// TwinCAT 3 PLC project PLC01
// ProgramVersion: 3.1.4023.0
// libraries:
//   Tc2_IoFunctions, * (Beckhoff Automation GmbH)
//   Tc2_Standard, * (Beckhoff Automation GmbH)
//   Tc2_System, * (Beckhoff Automation GmbH)
//   Tc2_Utilities, * (Beckhoff Automation GmbH)
//   Tc3_Module, * (Beckhoff Automation GmbH)
// project tree:
//   DUTs/Astrour/ FB_AstroUr.TcPOU
//   DUTs/Astrour/Functions/ fc_Day_Of_Year.TcPOU, fc_DEG.TcPOU, fc_DST.TcPOU, fc_Floor2.TcPOU, fc_Hour_To_Time.TcPOU, fc_Houre_To_TOD.TcPOU, fc_MODR.TcPOU, fc_RAD.TcPOU, fc_Set_Date.TcPOU, fc_Set_DT.TcPOU, fc_Sun_Midday.TcPOU, fc_Year_Of_Date.TcPOU
//   DUTs/Helgdag/ FB_SwedishHolidays.TcPOU
//   DUTs/Helgdag/Old/ FB_SwedishHolidaysOLD.TcPOU, POU_EasterDay.TcPOU
//   DUTs/KOH/ FB_KOH.TcPOU
//   DUTs/PID/ FB_PID.TcPOU
//   DUTs/Rampfunktion/ FB_Ramp.TcPOU
//   DUTs/Scale/ FB_Scale.TcPOU
//   DUTs/Select/ FB_Sel.TcPOU
//   DUTs/System/ FB_SystemTime.TcPOU, FB_TimerPulseSec.TcPOU, F_PLC_MS.TcPOU
//   DUTs/Tidkanal/ FB_TidKanalDrift.TcPOU
//   GVLs/ SYSTEM.TcGVL
//   / PlcTask.TcTTO
//   POUs/ MAIN.TcPOU
// real-time tasks:
//   TASK PlcTask: cycle T#10ms, priority 20, ADS port 350

CONFIGURATION PLC01
    RESOURCE PLC ON TwinCAT3
        TASK PlcTask(INTERVAL := T#10ms, PRIORITY := 20);
        PROGRAM MAIN WITH PlcTask : MAIN;
    END_RESOURCE
END_CONFIGURATION

// ---- GVLs/SYSTEM.TcGVL
{attribute 'qualified_only'}
VAR_GLOBAL
	nAliveCounter					: SINT; 			// PLC alive counter
    sDateAndTime					: STRING;			// Time and date
	dtSystemTime					: DATE_AND_TIME;	// Date and time
    uiYear							: UINT;				// Systemtime Year
    uiMonth							: UINT;				// Systemtime Month
    uiDayOfWeek 					: UINT;				// Systemtime Day of week
    uiDay							: UINT;				// Systemtime Day
    uiHour							: UINT;				// Systemtime Hour
    uiMinute						: UINT;				// Systemtime Minute
    uiSecond						: UINT;				// Systemtime Second
    uiMillisecond					: UINT;				// Systemtime Millisecond
    uiHourMinute					: UINT;				// Systemtime HourAndMinute
    dtDate							: DATE_AND_TIME;	// Variable for date and time
    uiTasktime						: UDINT;			// Tasktime
    uisystemtime 					: UDINT;			// System time	
    stTimeStruct					: TIMESTRUCT; 		// Timestruct
    sActTime						: STRING;			// Actual time
    uiSeconds						: UDINT;			// Variable for time in seconds
    bPowerFailDetect				: BOOL;				// Powerfail from UPS
    bIOError						: BOOL;				// IO-Error 
    bSavePersistentData				: BOOL;				// Saves persistent data manually              		
	tPlcUptime						: TIME;             // Last time PLC restart        		
	bWatchdogAlarm					: BOOL;				// Triggered watchdog alarm
	bWatchdogIsOK					: BOOL;				// Watchdog is ok  	
	bStartUp1s						: BOOL;				// Startup delay 1s after restart of TwinCAT
	bStartUp5s						: BOOL;				// Startup delay 5s after restart of TwinCAT
	bStartUp10s						: BOOL;				// Startup delay 10s after restart of TwinCAT
	bStartUp15s						: BOOL;				// Startup delay 15s after restart of TwinCAT
	bStartUp20s						: BOOL;				// Startup delay 20s after restart of TwinCAT
	bStartUp25s						: BOOL;				// Startup delay 25s after restart of TwinCAT
	bStartUp30s						: BOOL;				// Startup delay 30s after restart of TwinCAT
	bStartUp45s						: BOOL;				// Startup delay 45s after restart of TwinCAT
	bStartUp60s						: BOOL;				// Startup delay 60s after restart of TwinCAT
	bStartUp120s					: BOOL;				// Startup delay 120s after restart of TwinCAT
	bBurglarAlarmActive				: BOOL;				// Aktivt inbrottslarm 
	rOutdoorTemperature				: REAL;				// Outdoor temperature
	rAverageOutdoorTemperature		: REAL;				// Outdoor average temperature
	rAverageMinOutdoorTemperature	: REAL;				// Outdoor average min temperature	
	rAverageMaxOutdoorTemperature	: REAL;				// Outdoor average max temperature	
	rAverageIndoorTemperature		: REAL;				// Indoor average temperature
	bSummerCondition				: BOOL;        		// Summer condition active
	rCalculatedDewpoint				: REAL;				// Dewpoint   		          	

	sSystemID						: STRING;			// Current System ID
	sHostName						: STRING;			// Current hostname
	sAMSNetID						: STRING;			// Current AMS net ID
	sTargetType						: STRING;           
	sHardwareModel 					: STRING;
	sHardwareSerialNumber			: STRING;
	sHardwareVersion 				: STRING;
	sHardwareDate					: STRING;
	sHardwareCPU 					: STRING;
	sImageDevice					: STRING;
	sImageVersion 					: STRING;
	sImageLevel 					: STRING;
	sImageOsName 					: STRING;
	sImageOsVersion 				: STRING;
	sTwinCATVersion 				: STRING;
	sTwinCATRevision 				: STRING;
	sTwinCATBuild 					: STRING;
	sTwinCATLevel					: STRING;
	udiCpuUsage						: UDINT;	
	iArrWildCards					: ARRAY [0..100] OF INT;
	bArrWildCards					: ARRAY [0..100] OF BOOL;	
	
	
END_VAR

// ---- POUs/MAIN.TcPOU
PROGRAM MAIN
VAR
	fbTimeChannel 				: FB_TidkanalDrift;	
	fbAstroUr					: FB_AstroUr;
	fbSystemTime 				: FB_SystemTime;
	fbSwedishHolidays			: FB_SwedishHolidays;
	fbKOHFunction				: FB_KOH;
	
	bActivateTimeChannel		: BOOL; // Detta är en kommentar
	wMondayStartTime 			: WORD; // Detta är en kommentar
	wMondayStopTime 			: WORD; // Detta är en kommentar
	wTuesdayStartTime 			: WORD; // Detta är en kommentar
	wTuesdayStopTime 			: WORD; // Detta är en kommentar
	wWednesdayStartTime 		: WORD; // Detta är en kommentar
	wWednesdayStopTime 			: WORD; // Detta är en kommentar
	wThursdayStartTime 			: WORD; // Detta är en kommentar
	wThursdayStopTime 			: WORD; // Detta är en kommentar
	wFridayStartTime 			: WORD; // Detta är en kommentar
	wFridayStopTime 			: WORD; // Detta är en kommentar
	wSaturdayStartTime 			: WORD; // Detta är en kommentar
	wSaturdayStopTime 			: WORD; // Detta är en kommentar
	wSundayStartTime 			: WORD; // Detta är en kommentar
	wSundayStopTime 			: WORD; // Detta är en kommentar
	bTimeChannelActive			: BOOL; // Detta är en kommentar
	bSommarTidAktiv				: BOOL; // Detta är en kommentar
	bDetArMorktUteJustNu		: BOOL; // Detta är en kommentar
	strSoluppgang				: STRING; // Detta är en kommentar
	strSolnedgang				: STRING; // Detta är en kommentar
	//dActDate					: DATE:= D#2025-3-19; 
	dActDate					: DATE_AND_TIME; 
	dtTheDateAndTime			: DATE_AND_TIME;
	
	bLangfredagACT				: BOOL;
	bSkartorsdagACT				: BOOL;
	bPaskDagenACT				: BOOL;
	bPaskaftonACT				: BOOL;
	bAnnanDagPaskACT			: BOOL;
	bKristihimmelACT			: BOOL;
	bPingstAftonACT				: BOOL;
	bPingstDagenACT				: BOOL;
	bMidsommarDagenACT			: BOOL;
	bMidsommarAftonACT			: BOOL;
	bHalloweenACT				: BOOL;
	bJulaftonACT				: BOOL;
	bJuldagenACT				: BOOL;
	bAnnandagjulACT				: BOOL;
	bTrettondagACT				: BOOL;
	bNyarsaftonACT				: BOOL;
	bNyarsdagenACT				: BOOL;
	bForstamajACT				: BOOL;
	bNationaldagACT				: BOOL;
	bHelgDagAktivACT 			: BOOL;
	bAny						: BOOL; 
	iDay						: INT;
	
	// koh	
	bVarEnableKOHFunction		: BOOL;
	bVarBlockKOHFunction		: BOOL;
	bVarExceptionKOH			: BOOL;
	wVarMondayOn				: WORD;
	wVarMondayOff				: WORD;
	wVarTuesdayOn				: WORD;
	wVarTuesdayOff				: WORD;
	wVarWednesdayOn				: WORD;
	wVarWednesdayOff			: WORD;
	wVarThursdayOn				: WORD;
	wVarThursdayOff				: WORD;
	wVarFridayOn				: WORD;
	wVarFridayOff				: WORD;
	wVarSaturdayOn				: WORD;
	wVarSaturdayOff				: WORD;
	wVarSundayOn				: WORD;
	wVarSundayOff 				: WORD;
	diVarSystemCalcSetpoint 	: DINT;
	diVarDownRampTime  			: DINT;
	diVarSPEveningReduction 	: DINT;
	diVarSPWeekendReduction 	: DINT;
	diVarSPHolidayReduction 	: DINT;
	diVarSPExceptionReduction  	: DINT;
	diVarActualAverageRoomTemp 	: DINT;
	diVarAllowedMinRoomTemp  	: DINT;
	bVarKOHActive 				: BOOL;
	bVarKOHBlocked 				: BOOL;
	bVarAlarmBlocked			: BOOL;
	bVarAlarmMinTemp 			: BOOL;
	diVarKOHCalcOffset 			: DINT;
	bVarRampTimeActive			: BOOL;
	
END_VAR

VAR PERSISTENT	
	rLatitudeOrebro				: REAL; // Detta är en kommentar
	rLongitudeOrebro			: REAL; // Detta är en kommentar
	iOffsetSoluppgang			: INT; // Detta är en kommentar
	iOffsetSolnedgang			: INT; // Detta är en kommentar
END_VAR

fbSystemTime();
POU_EasterDay();

fbTimeChannel(
	bEn:= 					bActivateTimeChannel, 
	wMondayOn:= 			wMondayStartTime, 
	wMondayOff:= 			wMondayStopTime, 
	wTuesdayOn:= 			wTuesdayStartTime, 
	wTuesdayOff:= 			wTuesdayStopTime, 
	wWednesdayOn:= 			wWednesdayStartTime, 
	wWednesdayOff:= 		wWednesdayStopTime, 
	wThursdayOn:= 			wThursdayStartTime, 
	wThursdayOff:= 			wThursdayStopTime, 
	wFridayOn:= 			wFridayStartTime, 
	wFridayOff:= 			wFridayStopTime, 
	wSaturdayOn:= 			wSaturdayStartTime, 
	wSaturdayOff:= 			wSaturdayStopTime, 
	wSundayOn:= 			wSundayStartTime, 
	wSundayOff:= 			wSundayStopTime, 
	bOn=> 					bTimeChannelActive);

fbAstroUr(
	rLatitude:= 			rLatitudeOrebro, // Sätt latitud för platen du ska mäta på         
	rLongitude:= 			rLongitudeOrebro, // Sätt longitud för platsen du ska mäta på      
	iOffsetSunrise:= 		iOffsetSoluppgang, // Förskjut soluppgången här (teoretiskt)       
	iOffsetSunset:= 		iOffsetSolnedgang, // Förskjut solnedgången här (teoretiskt)       
	strSunrise=> 			strSoluppgang, // Detta är det förväntade klockslaget på soluppgång
	strSunset=> 			strSolnedgang, // Detta är det förväntade klockslaget på solnedgång
	bSummertime=> 			bSommarTidAktiv, // Det råder sommartid, åk till stranden          
	bDark=> 				bDetArMorktUteJustNu); // Är denna aktiv är det mörkt ute	         

fbSystemTime();
dActDate:=(fbSystemTime.dtSystemTime);

fbSwedishHolidays(
	dtActualDateAndTime=> 	dtTheDateAndTime, 
	bLangfredag=> 			bLangfredagACT, 
	bSkartorsdag=> 			bSkartorsdagACT, 
	bPaskDagen=> 			bPaskDagenACT, 
	bPaskafton=> 			bPaskaftonACT, 
	bAnnanDagPask=> 		bAnnanDagPaskACT, 
	bKristihimmel=> 		bKristihimmelACT, 
	bPingstAfton=> 			bPingstAftonACT, 
	bPingstDagen=> 			bPingstDagenACT, 
	bMidsommarDagen=> 		bMidsommarDagenACT, 
	bMidsommarAfton=> 		bMidsommarAftonACT, 
	bHalloween=> 			bHalloweenACT, 
	bJulafton=> 			bJulaftonACT, 
	bJuldagen=> 			bJuldagenACT, 
	bAnnandagjul=> 			bAnnandagjulACT, 
	bTrettondag=> 			bTrettondagACT, 
	bNyarsafton=> 			bNyarsaftonACT, 
	bNyarsdagen=> 			bNyarsdagenACT, 
	bForstamaj=> 			bForstamajACT, 
	bNationaldag=> 			bNationaldagACT, 
	bHelgDagAktiv=> 		bHelgDagAktivACT);


iDay:=fc_Day_Of_Year(IDATE:=TO_DATE (dActDate) );

	
	
fbKOHFunction(
	bEnableKOHFunction:= 			bVarEnableKOHFunction, 
	bBlockKOHFunction:= 			bVarBlockKOHFunction, 
	bExceptionKOH:= 				bVarExceptionKOH, 
	wMondayOn:= 					wVarMondayOn, 
	wMondayOff:= 					wVarMondayOff, 
	wTuesdayOn:= 					wVarTuesdayOn, 
	wTuesdayOff:= 					wVarTuesdayOff, 
	wWednesdayOn:= 					wVarWednesdayOn, 
	wWednesdayOff:= 				wVarWednesdayOff, 
	wThursdayOn:= 					wVarThursdayOn, 
	wThursdayOff:= 					wVarThursdayOff, 
	wFridayOn:= 					wVarFridayOn, 
	wFridayOff:= 					wVarFridayOff, 
	wSaturdayOn:= 					wVarSaturdayOn, 
	wSaturdayOff:= 					wVarSaturdayOff, 
	wSundayOn:= 					wVarSundayOn, 
	wSundayOff:= 					wVarSundayOff, 
	diSystemCalcSetpoint:= 			diVarSystemCalcSetpoint, 
	diDownRampTime:= 				diVarDownRampTime, 
	diSPEveningReduction:= 			diVarSPEveningReduction, 
	diSPWeekendReduction:= 			diVarSPWeekendReduction, 
	diSPHolidayReduction:= 			diVarSPHolidayReduction, 
	diSPExceptionReduction:= 		diVarSPExceptionReduction, 
	diActualAverageRoomTemp:= 		diVarActualAverageRoomTemp, 
	diAllowedMinRoomTemp:= 			diVarAllowedMinRoomTemp, 
	bKOHActive=> 					bVarKOHActive, 
	bKOHBlocked=> 					bVarKOHBlocked, 
	bAlarmBlocked=> 				bVarAlarmBlocked, 
	bAlarmMinTemp=> 				bVarAlarmMinTemp, 
	diKOHCalcOffset=> 				diVarKOHCalcOffset, 
	bRampTimeActive=> 				bVarRampTimeActive);

END_PROGRAM

// ---- DUTs/Tidkanal/FB_TidKanalDrift.TcPOU
FUNCTION_BLOCK FB_TidKanalDrift
VAR_INPUT
	bEn				: BOOL;		// Aktivera block
	wMondayOn		: WORD;		// Starttid Måndag
	wMondayOff		: WORD;		// Stopptid Måndag
	wTuesdayOn		: WORD;		// Starttid Tisdag
	wTuesdayOff		: WORD;		// Stopptid Tisdag
	wWednesdayOn	: WORD;		// Starttid Onsdag
	wWednesdayOff	: WORD;		// Stopptid Onsdag
	wThursdayOn		: WORD;		// Starttid Torsdag
	wThursdayOff	: WORD;		// Stopptid Torsdag
	wFridayOn		: WORD;		// Starttid Fredag
	wFridayOff		: WORD;		// Stopptid Fredag
	wSaturdayOn		: WORD;		// Starttid Lördag
	wSaturdayOff	: WORD;		// Stopptid Lördag
	wSundayOn		: WORD;		// Starttid Söndag
	wSundayOff		: WORD;		// Stopptid Söndag
END_VAR
	
VAR_OUTPUT
	bOn				: BOOL;		// Tidkanal aktiv
END_VAR


VAR
	fbSystemTime 	: FB_SystemTime;
END_VAR

// Tidkanal
fbSystemTime();
IF bEN THEN

CASE fbSystemTime.nWeekDay OF
	
		1: // Måndag 
		IF wMondayOff < wMondayOn THEN
			// 22:00-03:00
			IF fbSystemTime.nHourMinute >= wMondayOn OR fbSystemTime.nHourMinute < wMondayOff THEN
				bOn := TRUE;
			ELSE
				bOn := FALSE;
			END_IF
		ELSE
			// 06:00-22:00	
			IF fbSystemTime.nHourMinute >= wMondayOn AND fbSystemTime.nHourMinute < wMondayOff THEN
				bOn := TRUE;
			ELSE
				bOn := FALSE;
			END_IF
		END_IF	
		
		2: // Tisdag
		IF wTuesdayOff < wTuesdayOn THEN
			// 22:00-03:00
			IF fbSystemTime.nHourMinute >= wTuesdayOn OR fbSystemTime.nHourMinute < wTuesdayOff THEN
				bOn := TRUE;
			ELSE
				bOn := FALSE;
			END_IF
		ELSE
			// 06:00-22:00	
			IF fbSystemTime.nHourMinute >= wTuesdayOn AND fbSystemTime.nHourMinute < wTuesdayOff THEN
				bOn := TRUE;
			ELSE
				bOn := FALSE;
			END_IF
		END_IF		
		
		3: // Onsdag
		IF wWednesdayOff < wWednesdayOn THEN
			// 22:00-03:00
			IF fbSystemTime.nHourMinute >= wWednesdayOn OR fbSystemTime.nHourMinute < wWednesdayOff THEN
				bOn := TRUE;
			ELSE
				bOn := FALSE;
			END_IF
		ELSE
			// 06:00-22:00	
			IF fbSystemTime.nHourMinute >= wWednesdayOn AND fbSystemTime.nHourMinute < wWednesdayOff THEN
				bOn := TRUE;
			ELSE
				bOn := FALSE;
			END_IF
		END_IF	
		
		4: // Torsdag
		IF wThursdayOff < wThursdayOn THEN
			// 22:00-03:00
			IF fbSystemTime.nHourMinute >= wThursdayOn OR fbSystemTime.nHourMinute < wThursdayOff THEN
				bOn := TRUE;
			ELSE
				bOn := FALSE;
			END_IF
		ELSE
			// 06:00-22:00	
			IF fbSystemTime.nHourMinute >= wThursdayOn AND fbSystemTime.nHourMinute < wThursdayOff THEN
				bOn := TRUE;
			ELSE
				bOn := FALSE;
			END_IF
		END_IF	

		5: // Fredag 
		IF wFridayOff < wFridayOn THEN
			// 22:00-03:00
			IF fbSystemTime.nHourMinute >= wFridayOn OR fbSystemTime.nHourMinute < wFridayOff THEN
				bOn := TRUE;
			ELSE
				bOn := FALSE;
			END_IF
		ELSE
			// 06:00-22:00	
			IF fbSystemTime.nHourMinute >= wFridayOn AND fbSystemTime.nHourMinute < wFridayOff THEN
				bOn := TRUE;
			ELSE
				bOn := FALSE;
			END_IF
		END_IF	
		
		6: // Lördag
		IF wSaturdayOff < wSaturdayOn THEN
			// 22:00-03:00
			IF fbSystemTime.nHourMinute >= wSaturdayOn OR fbSystemTime.nHourMinute < wSaturdayOff THEN
				bOn := TRUE;
			ELSE
				bOn := FALSE;
			END_IF
		ELSE
			// 06:00-22:00	
			IF fbSystemTime.nHourMinute >= wSaturdayOn AND fbSystemTime.nHourMinute < wSaturdayOff THEN
				bOn := TRUE;
			ELSE
				bOn := FALSE;
			END_IF
		END_IF	
		
		0: // Söndag
		IF wSundayOff < wSundayOn THEN
			// 22:00-03:00
			IF fbSystemTime.nHourMinute >= wSundayOn OR fbSystemTime.nHourMinute < wSundayOff THEN
				bOn := TRUE;
			ELSE
				bOn := FALSE;
			END_IF
		ELSE
			// 06:00-22:00	
			IF fbSystemTime.nHourMinute >= wSundayOn AND fbSystemTime.nHourMinute < wSundayOff THEN
				bOn := TRUE;
			ELSE
				bOn := FALSE;
			END_IF
		END_IF
END_CASE


ELSE bOn := FALSE;
	
END_IF

END_FUNCTION_BLOCK

// ---- DUTs/System/FB_SystemTime.TcPOU
(*
:Beskrivning:	| Läser systemtiden.
:Instruktioner:	| Ändra sAMSNetID för annan tidsserver. Lämna tom för lokal tid i PLC.

:Versionshistorik:
+-------------+------------+----------------+------------+------------------------------------------+
|Datum        | Version    | Skapad under   | Författare | Kommentar                                |
+=============+============+================+============+==========================================+
|2020-02-20   | 1.0.0.1    | V3.1.4022.30   | CMC dev.   | Funktionsblock skapat                    |
+-------------+------------+----------------+------------+------------------------------------------+
	
*)
FUNCTION_BLOCK FB_SystemTime
VAR_INPUT
	sAMSNetID			: STRING:='';	// AMSNet-ID
END_VAR

VAR_OUTPUT
	dtSystemTime		: DT;			// Systemtid
	bGetTimeBusy		: BOOL;			// Busy  		
	bGetTimeError		: BOOL;			// Error
	nGetTimeErrorCode	: UDINT;		// ErrorID
	nYear				: DWORD;		// År
	nMonth				: DWORD;		// Månad
	nDay				: DWORD;		// Dag
	nWeekDay 			: DWORD;		// Veckodag
	nHour				: DWORD;		// Timme
	nMinute 			: DWORD;		// Minut
	nSecond				: DWORD;		// Sekund
	nMilliSecond		: DWORD;		// Millisekund
	nHourMinute			: DWORD;		// Timme och minut (HHMM)
END_VAR

VAR
	fbGetTime			: NT_GetTime;
	fbTimerPulseSec		: FB_TimerPulseSec;
END_VAR

fbTimerPulseSec(bStart := TRUE, nTime := 5); // FB_TimerPulseSec
fbGetTime(NETID := sAMSNetID, START := fbTimerPulseSec.bPulse, TMOUT := T#5s); // NT_GetTime
bGetTimeBusy := fbGetTime.BUSY;
bGetTimeError := fbGetTime.ERR;
nGetTimeErrorCode := fbGetTime.ERRID;
dtSystemTime := SYSTEMTIME_TO_DT(TIMESTR := fbGetTime.TIMESTR);
nYear := TO_DWORD(fbGetTime.TIMESTR.wYear);
nMonth := TO_DWORD(fbGetTime.TIMESTR.wMonth);
nDay := TO_DWORD(fbGetTime.TIMESTR.wDay);
nWeekDay := TO_DWORD(fbGetTime.TIMESTR.wDayOfWeek);
nHour := TO_DWORD(fbGetTime.TIMESTR.wHour);
nMinute := TO_DWORD(fbGetTime.TIMESTR.wMinute);
nSecond := TO_DWORD(fbGetTime.TIMESTR.wSecond);
nMilliSecond := TO_DWORD(fbGetTime.TIMESTR.wMilliseconds);
nHourMinute := nHour * 100 + nMinute;

END_FUNCTION_BLOCK

// ---- DUTs/System/FB_TimerPulseSec.TcPOU
(*
:Beskrivning:	| Timern är igång så länge bStart är hög. bPulse pulsar när bStart går från FALSE till TRUE och när nTIME är uppnådd. När nTIME är uppnådd börjar timern räkna om.
:Instruktioner:	|  

:Versionshistorik:
+-------------+------------+----------------+------------+------------------------------------------+
|Datum        | Version    | Skapad under   | Författare | Kommentar                                |
+=============+============+================+============+==========================================+
|2020-02-21   | 1.0.0.1    | V3.1.4022.30   | CMC dev.   | Funktionsblock skapat					|
+-------------+------------+----------------+------------+------------------------------------------+
	
*)
FUNCTION_BLOCK FB_TimerPulseSec
VAR_INPUT
	bStart 		: BOOL;  	// Aktivera timer
	nTIME		: DWORD; 	// Tid mellan pulserna (s)
END_VAR

VAR_OUTPUT
	bPulse		: BOOL; 	// Pulsutgång
END_VAR

VAR
	Start		: BOOL;
	init		: BOOL;
	tx			: DWORD;
	last		: DWORD;
	ms			: DWORD;
	Sec			: UDINT;
	
	R_TRIG		: R_TRIG;
END_VAR

(*

Information om block:

Källa: Oscat OnTime

*)

// Read system time
tx := F_PLC_MS();

// Make sure the first cycle works correctly
IF NOT init OR NOT bStart THEN
	init := TRUE;
	ms := 0;
ELSIF bStart THEN
	// Add the current milliseconds
	ms := (tx - last) + ms;
	IF ms >= 100 THEN
		Sec := Sec + 1;
		ms := ms - 100;
	END_IF
END_IF

IF NOT bStart THEN
	Sec := 0;
END_IF
last := tx;

IF bStart AND NOT Start THEN
	R_TRIG(CLK := bStart, Q => bPulse);
	Start := TRUE;
ELSIF bStart AND Sec >= TO_UDINT(nTIME) THEN
	bPulse := TRUE;
	Sec := 0;
ELSIF bStart THEN	
	bPulse := FALSE;
	Sec := Sec;
ELSE
	bPulse := FALSE;
	Start := FALSE;
	R_TRIG(CLK := FALSE);
END_IF

END_FUNCTION_BLOCK

// ---- DUTs/System/F_PLC_MS.TcPOU
(*
:Beskrivning:	| Hämtar PLCns interna timer i Millisekunder.
:Instruktioner:	|  

:Versionshistorik:
+-------------+------------+----------------+------------+-------------------------------------------+
|Datum        | Version    | Skapad under   | Författare | Kommentar                                 |
+=============+============+================+============+===========================================+
|2020-02-21   | 1.0.0.1    | V3.1.4022.30   | CMC dev.   | Funktion skapad							 |
+-------------+------------+----------------+------------+-------------------------------------------+
	
*)
FUNCTION F_PLC_MS : DWORD;	// Millisekunder
VAR CONSTANT
	N 			: INT := 0;
	debug		: BOOL := 0;
	offset		: DWORD := 0;
END_VAR
VAR
	tx		 	: TIME;		// Timer i Millisekunder
END_VAR

(*

Information om block:

Källa: Oscat T_PLC_MS

*)

tx := TIME();
F_PLC_MS := TIME_TO_DWORD(Tx);

IF debug THEN
	F_PLC_MS := (SHL(F_PLC_MS,N) OR SHL(DWORD#1,N)-1) + OFFSET;
END_IF;

END_FUNCTION

// ---- DUTs/Astrour/FB_AstroUr.TcPOU
FUNCTION_BLOCK FB_AstroUr

VAR_INPUT
	rLatitude 				: REAL; // Latitud där anläggningen befinner sig
	rLongitude 				: REAL; // Longitud där anläggningen befinner sig
	iOffsetSunrise			: DINT;	// Offset för soluppgång i minuter
	iOffsetSunset			: DINT;	// Offset för solnedgång i minuter
END_VAR         			
                			
VAR_OUTPUT      			
	strSunrise				: STRING(5); // SunRise som string
	strSunset				: STRING(5); // Sunset som string
	bSummertime				: BOOL; // Indikering sommartid
	bDark					: BOOL; // Indikering solen har gått ner
END_VAR

VAR
	fbSystemTime 			: FB_SystemTime;
	                		
	dDate 					: DATE; // Aktuellt datum
	rSunPosMidday			: REAL; // Solens position mitt på dagen
	tDelta					: TIME; // Dela, tiden från mitt på dagen till soluppgång/nedgång
	rLatRad					: REAL; // Latitud omberäknad till radianer
	todActSunRise 			: TOD; // Soluppgång aktuell dag
	todActSunSet 			: TOD; // Solnedgång aktuell dag
	todActTime				: TIME_OF_DAY; // Aktuellt klockslag	
	todMidDay				: TOD; // Aktuell middagstid (när solen står i Zenit)
	rSunAngleMidday 		: REAL; // Solens vinkel mitt på dagen	
	dwSunSet				: DWORD; // Mellanvariabel för konvertering
	dwSunRise				: DWORD; // Mellanvariabel för konvertering            	
	rHeightAngle			: REAL := -0.83333333333; // Solens tim-vinkel
	todSunRise				: TOD;
	todSunSet				: TOD;
	dtVarSystemTime 		: DATE_AND_TIME;
	todVarTimeOfDay			: TIME_OF_DAY;
	
	dwSunRiseMinute			: DWORD;
	dwSunRiseHour			: DWORD;
	dwSunRiseTime			: DWORD;
	
	dwSunSetMinute			: DWORD;
	dwSunSetHour			: DWORD;
	dwSunSetTime			: DWORD;
	
	strHourSunRise			: STRING(2);
	strMinuteSunRise		: STRING(2);  
	strHourSunSet			: STRING(2);
	strMinuteSunSet			: STRING(2);   
END_VAR

// Anrop och variabelhanteringar
fbSystemTime();

dtVarSystemTime:= 	fbSystemTime.dtSystemTime;
todActTime:= 		todVarTimeOfDay;
dDate:= 			TO_DATE(dtVarSystemTime);
todVarTimeOfDay:= 	TO_TOD (fbSystemTime.dtSystemTime); 
rLatRad:=			rLatitude * 0.0174532925199433;
todMidDay:=			fc_Sun_Midday(rLongitude, dDate);

// Beräknar solposition
rSunPosMidday := 0.40954 * SIN(0.0172 * (INT_TO_REAL(fc_Day_Of_Year(dDate)) - 79.35));
rSunAngleMidday := fc_DEG(rSunPosMidday);

// Sätter solvinkel
IF rSunAngleMidday > 180.0 THEN
	rSunAngleMidday := rSunAngleMidday - 360.0;
END_IF;

rSunAngleMidday := 90.0 - rLatitude + rSunAngleMidday;

// Beräknar tid mellan solens högsta punkt och solnedgång resp. soluppgång
tDelta := fc_Hour_To_Time(ACOS((SIN(fc_RAD(rHeightAngle)) - SIN(rLatRad) * SIN(rSunPosMidday)) / (COS(rLatRad) * COS(rSunPosMidday))) * 3.819718632);

todActSunRise := todMidDay - tDelta;
todActSunSet := todMidDay + tDelta;

// Sommartid eller ej 
bSummertime := fc_DST(UTC:= dtVarSystemTime);

// Förskjutning om sommartid råder
IF bSummertime THEN
	todSunRise 	:= todActSunRise + T#2H + DINT_TO_TIME(iOffsetSunrise * 60000);
	todSunSet	:= todActSunSet  + T#2H + DINT_TO_TIME(iOffsetSunset  * 60000); ELSE
	todSunRise 	:= todActSunRise + T#1H + DINT_TO_TIME(iOffsetSunrise * 60000);
	todSunSet	:= todActSunSet  + T#1H + DINT_TO_TIME(iOffsetSunset  * 60000);
END_IF

// Sätter bool om det är mörkt ute
IF (todSunRise > todActTime) OR (todSunSet < todActTime) THEN
	bDark := TRUE; ELSE
	bDark := FALSE;	
END_IF

// Skapar STRING för att presentera soluppgång / solnedgång i SCADA/KOD

// Soluppgång
dwSunRiseHour:= TOD_TO_DWORD(todSunRise)/3600000;
dwSunRiseMinute:= TOD_TO_DWORD(todSunRise)/60000;
dwSunRiseTime:= dwSunRiseMinute -(60 * dwSunRiseHour);

IF dwSunRiseHour < 10 THEN
	strHourSunRise := concat ('0',DWORD_TO_STRING(dwSunRiseHour)); ELSE
	strHourSunRise := DWORD_TO_STRING(dwSunRiseHour);	
END_IF

IF dwSunRiseTime < 10 THEN 
	strMinuteSunRise := concat('0',DWORD_TO_STRING(dwSunRiseTime)); ELSE
	strMinuteSunRise := DWORD_TO_STRING(dwSunRiseTime);
END_IF

// Solnedgång
dwSunSetHour:= TOD_TO_DWORD(todSunSet)/3600000;
dwSunSetMinute:= TOD_TO_DWORD(todSunSet)/60000;
dwSunSetTime:= dwSunSetMinute -(60 * dwSunSetHour);

IF dwSunSetHour < 10 THEN
	strHourSunSet := concat ('0',DWORD_TO_STRING(dwSunSetHour)); ELSE
	strHourSunSet := DWORD_TO_STRING(dwSunSetHour);	
END_IF

IF dwSunSetMinute < 10 THEN 
	strMinuteSunSet := concat('0',DWORD_TO_STRING(dwSunSetTime)); ELSE
	strMinuteSunSet := DWORD_TO_STRING(dwSunSetTime);
END_IF

// Klara strängar
strSunRise:= concat(strHourSunRise,':');
strSunRise:= concat(strSunRise, strMinuteSunRise);
strSunSet:= concat(strHourSunSet,':');
strSunSet:= concat(strSunSet, strMinuteSunSet);

END_FUNCTION_BLOCK

// ---- DUTs/Astrour/Functions/fc_Sun_Midday.TcPOU
FUNCTION fc_Sun_Midday : TOD
VAR_INPUT
	LON : REAL;
	UTC : DATE;
END_VAR
VAR
	T 		: REAL;
	OFFSET 	: REAL;
END_VAR

T := INT_TO_REAL(fc_Day_Of_Year(utc));


OFFSET := -0.1752 * SIN(0.033430 * T + 0.5474) - 0.1340 * SIN(0.018234 * T - 0.1939);
fc_Sun_Midday := fc_Houre_To_TOD(12.0 - OFFSET - lon * 0.0666666666666);

END_FUNCTION

// ---- DUTs/Astrour/Functions/fc_Day_Of_Year.TcPOU
FUNCTION fc_Day_Of_Year : int
VAR_INPUT
		IDATE : DATE;
END_VAR
VAR
END_VAR


fc_Day_Of_Year := UDINT_TO_INT((DATE_TO_UDINT(idate) / UDINT#86400) MOD UDINT#1461);

IF fc_Day_Of_Year > 729 THEN
	IF fc_Day_Of_Year > 1095 THEN fc_Day_Of_Year := fc_Day_Of_Year - 1095; ELSE fc_Day_Of_Year := fc_Day_Of_Year - 729; END_IF;
ELSIF fc_Day_Of_Year > 364 THEN
	fc_Day_Of_Year := fc_Day_Of_Year - 364;
ELSE
	fc_Day_Of_Year := fc_Day_Of_Year + 1;
END_IF;

END_FUNCTION

// ---- DUTs/Astrour/Functions/fc_Houre_To_TOD.TcPOU
FUNCTION fc_Houre_To_TOD : TOD
VAR_INPUT
		IN : REAL;
END_VAR
VAR
END_VAR

fc_Houre_To_TOD := DWORD_TO_TOD(REAL_TO_DWORD(IN * 3600000));

END_FUNCTION

// ---- DUTs/Astrour/Functions/fc_DEG.TcPOU
FUNCTION fc_DEG : real
VAR_INPUT
		rad : REAL;
END_VAR
VAR
END_VAR

fc_DEG := fc_MODR(57.29577951308232 * RAD, 360.0);

END_FUNCTION

// ---- DUTs/Astrour/Functions/fc_MODR.TcPOU
FUNCTION fc_MODR : real
VAR_INPUT
	IN : REAL;
	DIVI : REAL;
END_VAR
VAR
END_VAR

IF divi = 0.0 THEN
	fc_MODR := 0.0;
ELSE
	fc_MODR := in - DINT_TO_REAL(fc_Floor2(in / divi)) * divi;
END_IF;

END_FUNCTION

// ---- DUTs/Astrour/Functions/fc_Floor2.TcPOU
FUNCTION fc_Floor2 : DINT
VAR_INPUT
	X : REAL;
END_VAR
VAR
END_VAR

fc_Floor2 := REAL_TO_DINT(X);
IF DINT_TO_REAL(fc_Floor2) > X THEN
	fc_Floor2 := fc_Floor2 - 1;
END_IF;

END_FUNCTION

// ---- DUTs/Astrour/Functions/fc_Hour_To_Time.TcPOU
FUNCTION fc_Hour_To_Time : Time
VAR_INPUT
		IN : REAL;
END_VAR
VAR
END_VAR

fc_Hour_To_Time := DWORD_TO_TIME(REAL_TO_DWORD(IN * 3600000));

END_FUNCTION

// ---- DUTs/Astrour/Functions/fc_RAD.TcPOU
FUNCTION fc_RAD : real
VAR_INPUT
	DEG : REAL;
END_VAR
VAR
END_VAR

fc_RAD := fc_MODR(0.0174532925199433 * DEG, 6.28318530717958647692528676655900576);

END_FUNCTION

// ---- DUTs/Astrour/Functions/fc_DST.TcPOU
FUNCTION fc_DST : bool
VAR_INPUT
	UTC 	: DT;
END_VAR
VAR
	yr 		: INT;
	yr4 	: DWORD;
	ltc		: DWORD;
	idate 	: DWORD;
END_VAR

yr := fc_Year_Of_Date(DT_TO_DATE(UTC));
ltc := DT_TO_DWORD(UTC);
idate := DT_TO_DWORD(fc_Set_DT(yr, 3, 31, 1, 0, 0));
yr4 := SHR(5 * INT_TO_DWORD(yr), 2) + 1;
fc_DST := (idate - ((yr4 + 3) MOD 7) * 86400 <= ltc) AND (idate + (214 - (yr4) MOD 7) * 86400 > ltc);

END_FUNCTION

// ---- DUTs/Astrour/Functions/fc_Year_Of_Date.TcPOU
FUNCTION fc_Year_Of_Date : INT
VAR_INPUT
		IDATE : DATE;
END_VAR
VAR
END_VAR

fc_Year_Of_Date := DWORD_TO_INT((DATE_TO_DWORD(idate) + 43200) / 31557600 + 1970);

END_FUNCTION

// ---- DUTs/Astrour/Functions/fc_Set_DT.TcPOU
FUNCTION fc_Set_DT : DT
VAR_INPUT
	year 	: INT;
	month 	: INT;
	day 	: INT;
	hour 	: INT;
	minute 	: INT;
	second 	: INT;
END_VAR
VAR
END_VAR

fc_Set_DT := DWORD_TO_DT(DATE_TO_DWORD(fc_Set_Date(YEAR, MONTH, day)) + INT_TO_DWORD(SECOND) + INT_TO_DWORD(MINUTE) * 60 + INT_TO_DWORD(HOUR) * 3600);

END_FUNCTION

// ---- DUTs/Astrour/Functions/fc_Set_Date.TcPOU
FUNCTION fc_Set_Date : date
VAR_INPUT
	YEAR 	: INT;
	MONTH 	: INT;
	DAY 	: INT;
END_VAR
VAR
	count 	: INT;
END_VAR

IF month > 2 THEN
	count := (month - 1) * 30;
	IF month > 7 THEN count := count + SHR(month - 3,1); ELSE count := count + SHR(month - 4,1); END_IF;
	(* chech for leap year and add one day if true *)
	IF SHL(year,14) = 0 THEN count := count + 1; END_IF;
ELSE
	count := (month - 1) * 31;
END_IF;

fc_Set_Date := DWORD_TO_DATE((INT_TO_DWORD(count + day - 1) + SHR(INT_TO_DWORD(year) * 1461 - 2878169, 2)) * 86400);

END_FUNCTION

// ---- DUTs/Helgdag/FB_SwedishHolidays.TcPOU
FUNCTION_BLOCK FB_SwedishHolidays
VAR_INPUT
END_VAR

VAR_OUTPUT
	dtActualDateAndTime			: DATE_AND_TIME;
	bLangfredag					: BOOL;
	bSkartorsdag				: BOOL;
	bPaskDagen					: BOOL;
    bPaskafton					: BOOL;
    bAnnanDagPask				: BOOL;
    bKristihimmel				: BOOL;
    bPingstAfton				: BOOL;
    bPingstDagen				: BOOL;
    bMidsommarDagen				: BOOL;
    bMidsommarAfton				: BOOL;
    bHalloween					: BOOL;
    bJulafton					: BOOL;
    bJuldagen					: BOOL;
    bAnnandagjul				: BOOL;
    bTrettondag					: BOOL;
    bNyarsafton					: BOOL;
    bNyarsdagen					: BOOL;
    bForstamaj					: BOOL;
    bNationaldag				: BOOL;
	bHelgDagAktiv				: BOOL;
END_VAR

VAR
	fbSystemTime 				: FB_SystemTime;
    iYear 						: INT; // Aktuellt år	
    iMonth						: INT;
	iDay						: INT;
    iEastermDayOfYear			: INT; // Påskdagens dagnummer i året
    isLeapYear 					: BOOL; // Flagga för skottår	
	stSystemTime				: TIMESTRUCT;
    arrMonthDays 				: ARRAY[1..12] OF INT := [31,28,31,30,31,30,31,31,30,31,30,31]; // Dagar per månad
    iDayOfYear					: INT;
    a, b, c, d, e, f, g, h, i, k, L, m, n : INT; // Variabler för Gauss algoritm
	iDayOfWeek					: INT;
	iActMonth					: INT;
	
	iVarHalloweenDay			: INT;
	iVarMidsommardagen 			: INT;
	iMidsommardagenDayOfYear	: INT;
	iVarMidsommardagenDayOfWeek	: INT;
	iVarMidsommardagen1			: INT;
	iSumDays					: INT;
	iVarDayOfYearCristmas		: INT;
	iVarDayForstamaj			: INT;
	iVarNationaldag				: INT;
	iVarJuldagen				: INT;
	
	iLangfredag					: INT;
 	iSkartorsdag				: INT;
	iPaskDagen					: INT;
 	iPaskafton					: INT;
 	iAnnanDagPask				: INT;
	iKristihimmel				: INT;
	iPingstAfton				: INT;
	iPingstDagen				: INT;
	iMidsommarDagen				: INT;
	iMidsommarAfton				: INT;
	iHalloween					: INT;
	iJulafton					: INT;
	iJuldagen					: INT;
	iAnnandagjul				: INT;
	iTrettondag					: INT;
    iNyarsafton					: INT;	
    iNyarsdagen					: INT;	
    iForstamaj					: INT;		
    iNationaldag				: INT;
END_VAR

VAR PERSISTENT
	iYear2000		: INT:=2000;
END_VAR

fbSystemTime();
iDayOfYear:= fc_Day_Of_Year(IDATE:=TO_DATE (fbSystemTime.dtSystemTime)) + 1;
iYear:= DWORD_TO_INT(fbSystemTime.nYear);
iDayOfWeek:= DWORD_TO_INT(fbSystemTime.nDay);
iActMonth:= TO_INT (fbSystemTime.nMonth);
dtActualDateAndTime:= (fbSystemTime.dtSystemTime);

// Gauss algoritm för att räkna ut påskdagen
a := iYear MOD 19;
b := iYear / 100;
c := iYear MOD 100;
d := b / 4;
e := b MOD 4;
f := (b + 8) / 25;
g := (b - f + 1) / 3;
h := (19 * a + b - d - g + 15) MOD 30;
i := c / 4;
k := c MOD 4;
L := (32 + 2 * e + 2 * i - h - k) MOD 7;
m := (a + 11 * h + 22 * L) / 451;
n := (h + L - 7 * m + 114);
iMonth := n / 31;
iDay := (n MOD 31) + 1;

// Kontrollera om året är skottår
IF (iYear MOD 4 = 0 AND iYear MOD 100 <> 0) OR (iYear MOD 400 = 0) THEN
    isLeapYear := TRUE;
    arrMonthDays[2] := 29; // Februari har 29 dagar i skottår
ELSE
    isLeapYear := FALSE;
END_IF

// Beräkna årets dag för påskdagen
iEastermDayOfYear := iDay; // Startvärde
FOR i := 1 TO iMonth - 1 DO
    iEastermDayOfYear := iEastermDayOfYear + arrMonthDays[i]; // Addera dagar i tidigare månader
END_FOR

// Beräkna årets dag för 31 oktober, Halloween
iVarHalloweenDay := 31; // Startvärde för Halloweens dag i oktober
FOR i := 1 TO 9 DO // Loopar igenom månaderna januari-september
    iVarHalloweenDay := iVarHalloweenDay + arrMonthDays[i]; // Addera dagar i tidigare månader
END_FOR


// 1. Beräkna veckodag för 20 juni enligt Zeller's Congruence
iVarMidsommardagenDayOfWeek := (20 + ((13 * 7) / 5) + (iYear MOD 100) + ((iYear MOD 100) / 4) + ((iYear / 100) / 4) - (2 * (iYear / 100))) MOD 7;

// 2. Konvertera från Zeller-format till Beckhoff-format (Söndag = 0, Måndag = 1, ..., Lördag = 6)
iVarMidsommardagenDayOfWeek := (iVarMidsommardagenDayOfWeek + 6) MOD 7;

// 3. Hitta första lördagen från och med 20 juni
IF iVarMidsommardagenDayOfWeek = 6 THEN
    iVarMidsommardagen := 20; // 20 juni är lördag
ELSE
    iVarMidsommardagen := 20 + ((6 - iVarMidsommardagenDayOfWeek) MOD 7);
END_IF

// 4. Beräkna årets dag (julianska kalenderdagar) inklusive skottår
iVarMidsommardagen1 := iVarMidsommardagen;

// Lägg till dagarna från januari till maj
iSumDays := 0;
FOR i := 1 TO 5 DO
    iSumDays := iSumDays + arrMonthDays[i];
END_FOR

// Om det är skottår, lägg till 1 dag efter februari
IF ((iYear MOD 4 = 0 AND iYear MOD 100 <> 0) OR (iYear MOD 400 = 0)) THEN
    iSumDays := iSumDays + 1;  // Flytta till här!
END_IF

iVarMidsommardagen1 := iVarMidsommardagen1 + iSumDays;


// Beräknar årets dag för 25 december
iVarDayOfYearCristmas := 24; // Startvärde för juldagen
FOR i := 1 TO 11 DO // Loopar igenom månaderna januari-november
    iVarDayOfYearCristmas := iVarDayOfYearCristmas + arrMonthDays[i]; // Addera dagar i tidigare månader
END_FOR

IF isLeapYear THEN
    iVarDayOfYearCristmas := iVarDayOfYearCristmas + 1;
END_IF

// Beräknar årets dag för 1 maj
iVarDayForstamaj := 0; // Startvärde för 1 maj
FOR i := 1 TO 4 DO // Loopar igenom månaderna januari-april *)
    iVarDayForstamaj := iVarDayForstamaj + arrMonthDays[i]; //Addera dagar i tidigare månader
END_FOR

IF isLeapYear THEN
    iVarDayForstamaj := iVarDayForstamaj + 1;
END_IF

// Beräkna sveriges nationaldag
iVarNationaldag := 5; // Startvärde för 6 juni
FOR i := 1 TO 5 DO // Loopar igenom månaderna januari-maj
    iVarNationaldag := iVarNationaldag + arrMonthDays[i]; // Addera dagar i tidigare månader
END_FOR
IF isLeapYear THEN
    iVarNationaldag := iVarNationaldag + 1;
END_IF


// Ger var värde för resp. dag
iLangfredag 		:= iEastermDayOfYear - 2;
iSkartorsdag	 	:= iEastermDayOfYear - 3;
iPaskDagen			:= iEastermDayOfYear;
iPaskafton 			:= iEastermDayOfYear - 1; 
iAnnanDagPask 		:= iEastermDayOfYear + 1; 
iKristihimmel 		:= iEastermDayOfYear + 39; 
iPingstAfton		:= iEastermDayOfYear + 48; 
iPingstDagen		:= iEastermDayOfYear + 49;
iMidsommarDagen		:= iVarMidsommardagen1;
iMidsommarAfton		:= iVarMidsommardagen1 - 1;
iHalloween			:= iVarHalloweenDay;
iJulafton			:= iVarDayOfYearCristmas - 1;
iJuldagen			:= iVarDayOfYearCristmas;
iAnnandagjul		:= iVarDayOfYearCristmas + 1;
iTrettondag			:= 6;
iNyarsafton			:= iVarDayOfYearCristmas + 6;
iNyarsdagen			:= 1; 
iForstamaj			:= iVarDayForstamaj;
iNationaldag		:= iVarNationaldag;

// Sätter bool för resp. dag
bLangfredag 		:= (iDayOfYear = (iLangfredag));
bSkartorsdag	 	:= (iDayOfYear = (iSkartorsdag));
bPaskDagen			:= (iDayOfYear = (iPaskDagen));
bPaskafton 			:= (iDayOfYear = (iPaskafton));
bAnnanDagPask 		:= (iDayOfYear = (iAnnanDagPask));
bKristihimmel 		:= (iDayOfYear = (iKristihimmel));
bPingstAfton		:= (iDayOfYear = (iPingstAfton));
bPingstDagen		:= (iDayOfYear = (iPingstDagen));
bHalloween			:= (iDayOfYear = (iHalloween));
bJulafton			:= (iDayOfYear = (iJulafton));
bJuldagen			:= (iDayOfYear = (iJuldagen));
bAnnandagjul		:= (iDayOfYear = (iAnnandagjul));
bTrettondag			:= (iDayOfYear = (iTrettondag));
bNyarsafton			:= (iDayOfYear = (iNyarsafton));
bNyarsdagen			:= (iDayOfYear = (iNyarsdagen));
bForstamaj			:= (iDayOfYear = (iForstamaj));
bNationaldag		:= (iDayOfYear = (iNationaldag));
bMidsommarDagen		:= (iDayOfYear = (iVarMidsommardagen1));
bMidsommarAfton		:= (iDayOfYear = (iVarMidsommardagen1)-1);

IF bLangfredag OR bSkartorsdag OR bPaskDagen OR	bPaskafton OR bAnnanDagPask OR bKristihimmel OR	bPingstAfton OR	bPingstDagen OR	bMidsommarDagen OR bMidsommarAfton OR bHalloween OR	bJulafton OR bJuldagen OR bAnnandagjul OR bTrettondag OR bNyarsafton OR	bNyarsdagen OR bForstamaj OR bNationaldag THEN
bHelgDagAktiv:= TRUE; ELSE
bHelgDagAktiv:= FALSE;
END_IF

END_FUNCTION_BLOCK

// ---- DUTs/KOH/FB_KOH.TcPOU
FUNCTION_BLOCK FB_KOH

VAR_INPUT
	bEnableKOHFunction				: BOOL; // Aktiverar KOH via driftindikering av VS-pump
	bBlockKOHFunction				: BOOL; // Blockera KOH via annan källa		
	bExceptionKOH					: BOOL; // Aktiverar undantags-funktion		
    wMondayOn						: WORD; // Tillslagstid för måndag [0000-2400]
    wMondayOff						: WORD; // Frånslagstid för måndag [0000-2400]
    wTuesdayOn						: WORD; // Tillslagstid för tisdag [0000-2400]
    wTuesdayOff						: WORD; // Frånslagstid för tisdag [0000-2400]
    wWednesdayOn					: WORD; // Tillslagstid för onsdag [0000-2400]
    wWednesdayOff					: WORD; // Frånslagstid för onsdag [0000-2400]
    wThursdayOn						: WORD; // Tillslagstid för torsdag [0000-2400]
    wThursdayOff					: WORD; // Frånslagstid för torsdag [0000-2400]
    wFridayOn						: WORD; // Tillslagstid för fredag [0000-2400]
    wFridayOff						: WORD; // Frånslagstid för fredag [0000-2400]
    wSaturdayOn						: WORD; // Tillslagstid för lördag [0000-2400]
    wSaturdayOff					: WORD; // Frånslagstid för lördag [0000-2400]
    wSundayOn						: WORD; // Tillslagstid för söndag [0000-2400]
    wSundayOff						: WORD; // Frånslagstid för söndag [0000-2400]
	
	diSystemCalcSetpoint			: DINT; // Systemets aktuella beräknade börvärde [0000-2400]
	diDownRampTime					: DINT; // Upprampning av förskjutning tillbaka till ursprungsberäkning av börvärde [0-1000 minuter (0-100)]
	diSPEveningReduction			: DINT; // Inställning börvärdessänka kvällstid måndag-söndag [0-1000 (0-100°C)]
	diSPWeekendReduction			: DINT; // Inställning börvärdessänka helgtid [0-1000 (0-100°C)]
	diSPHolidayReduction			: DINT; // Inställning börvärdessänka helgdagar [0-1000 (0-100°C)]
	diSPExceptionReduction			: DINT; // Inställning börvärdessänka undantagssänka [0-1000 (0-100°C)]
	diActualAverageRoomTemp			: DINT; // Aktuellt medelvärde rumstemperatur
	diAllowedMinRoomTemp			: DINT; // Lägsta tillåtna rumsmedeltemperatur [0-1000 (0-100°C)]
END_VAR

VAR_OUTPUT	
	bKOHActive						: BOOL; // KOH-funktion aktiv
	bKOHBlocked						: BOOL; // KOH-funktion blockerad från annan källa
	bAlarmBlocked					: BOOL; // Alarm, KOH-funktion blockerad [B]
	bAlarmMinTemp					: BOOL; // Lägsta rumstemperaturen uppnådd [B]
	diKOHCalcOffset					: DINT; // Aktuellt nytt beräknat börvärde
	bRampTimeActive					: BOOL; // Ramp-funktion aktiv
END_VAR

VAR
// Sytemtid	
	fbSystemTime 					: FB_SystemTime;
// Funktionsblock
	fbTidkanalKOH					: FB_TidKanalDrift; // Tidkanalsblock
	fbSwedishHolidays				: FB_SwedishHolidays; // Block för beräkning av svenska helgdagar
	fbRamp							: FB_Ramp; // Rampblock
	fbSel							: FB_Sel; // Selectblock av korrekt förskjutning
	fbPIDCascade					: FB_PID; // PID för kaskad av förskjutning

// Lokala variabler	
	bVarTidKanalAktiv				: BOOL; // Lokal variabel, tidkanal för drift aktiv
	dActDate						: DATE_AND_TIME; 	
	dtVarSystemTime 				: DATE_AND_TIME;
	todVarTimeOfDay					: TIME_OF_DAY;
	dDate 							: DATE; // Aktuellt datum
	todActTime						: TIME_OF_DAY; // Aktuellt klockslag
	iVarActDay						: INT; // Lokal variabel, aktuell dag. Måndag=1, Tisdag=2, Onsdag=3, Torsdag=4, Fredag=5, Lördag=6, Söndag=0
	bVarVardagAct					: BOOL; // Lokal variabel, Måndag-fredag aktiv
	bVarVeckoslutAct				: BOOL; // Lokal variabel, vanlig lördag-söndag aktiv
	bVarHelgdagAktiv				: BOOL; // Lokal variabel, någon helgdag är aktiv
	bVarExceptionAct				: BOOL; // Lokal variabel, undantagssänka aktiv
	
	bVarTKVardagAct					: BOOL; // Lokal variabel, Måndag-fredag aktiv
	bVarTKVeckoslutAct				: BOOL; // Lokal variabel, vanlig lördag-söndag aktiv
	bVarTKExceptionAct				: BOOL; // Lokal variabel, undantagssänka aktiv
	
	diVarSelOutPut					: DINT; // Lokal variabel, temp-värde
	diVarOffsetValue				: DINT; // Lokal variabel, värde som ska förskjuta beräknat börvärde
END_VAR

fbSystemTime();
dtVarSystemTime:= 	fbSystemTime.dtSystemTime;
todActTime:= 		todVarTimeOfDay;
dDate:= 			TO_DATE(dtVarSystemTime);
todVarTimeOfDay:= 	TO_TOD (fbSystemTime.dtSystemTime); 
// Kör hela KOH om det inte är blockerat
IF NOT bBlockKOHFunction THEN

//===========Startar KOH om pumpen för värmesystemet är i drift===========//
IF bEnableKOHFunction THEN

//===========Block för att beräkna svenska helgdagar===========//	
fbSwedishHolidays();

//===========Tidkanal för aktivering av KOH===========//
fbTidkanalKOH(
	bEn:= 						,
	wMondayOn:= 				wMondayOn,
	wMondayOff:= 				wMondayOff,
	wTuesdayOn:= 				wTuesdayOn,
	wTuesdayOff:= 				wTuesdayOff,
	wWednesdayOn:= 				wWednesdayOn,
	wWednesdayOff:= 			wWednesdayOff,
	wThursdayOn:= 				wThursdayOn,
	wThursdayOff:= 				wThursdayOff,
	wFridayOn:= 				wFridayOn,
	wFridayOff:= 				wFridayOff,
	wSaturdayOn:= 				wSaturdayOn,
	wSaturdayOff:= 				wSaturdayOff,
	wSundayOn:= 				wSundayOn,
	wSundayOff:= 				wSundayOff,
	bOn=> 						bVarTidKanalAktiv);
	
//=========== Aktiverar mån-fre, lör-sön, helgdag, undantag i fallande prio===========//
// Beräknar dag 0-6 
iVarActDay:=fc_Day_Of_Year(IDATE:=TO_DATE (dDate));
// Beräknar mån-fre 1-5
IF (iVarActDay >0 AND iVarActDay <5) AND NOT bVarHelgdagAktiv THEN
	bVarVardagAct:= TRUE;	
// Beräknar lör-sön 6,0
ELSIF (iVarActDay = 7 OR iVarActDay = 0) AND NOT bVarHelgdagAktiv THEN
	bVarVardagAct	:= FALSE;	
	bVarVeckoslutAct:= TRUE;
	bVarHelgdagAktiv:= FALSE;
	bVarExceptionAct:= FALSE;	
// Beräknar helgdag
ELSIF fbSwedishHolidays.bHelgDagAktiv THEN
	bVarVardagAct	:= FALSE;	
	bVarVeckoslutAct:= FALSE;
	bVarHelgdagAktiv:= TRUE;
	bVarExceptionAct:= FALSE;
// Beräknar undantag
ELSIF bExceptionKOH THEN
	bVarVardagAct	:= FALSE;	
	bVarVeckoslutAct:= FALSE;
	bVarHelgdagAktiv:= FALSE;
	bVarExceptionAct:= TRUE;
ELSE
	bVarVardagAct	:= FALSE;	
	bVarVeckoslutAct:= FALSE;
	bVarHelgdagAktiv:= FALSE;
	bVarExceptionAct:= FALSE;
END_IF


// Startar KOH via tidkanal och aktuellt veckoläge
IF bVarTidKanalAktiv AND bVarVardagAct THEN
	bVarTKVardagAct:=	 	TRUE;
	bVarTKVeckoslutAct:= 	FALSE;
	bVarHelgdagAktiv:=	 	FALSE;
	bVarTKExceptionAct:= 	FALSE;
ELSIF bVarTidKanalAktiv AND bVarVeckoslutAct THEN	
	bVarTKVardagAct:= 		FALSE;
	bVarTKVeckoslutAct:= 	TRUE;
	bVarHelgdagAktiv:= 		FALSE;
	bVarTKExceptionAct:= 	FALSE;
ELSIF bVarTidKanalAktiv AND bVarHelgdagAktiv THEN	
	bVarTKVardagAct:= 		FALSE;
	bVarTKVeckoslutAct:= 	FALSE;
	bVarHelgdagAktiv:= 		TRUE;
	bVarTKExceptionAct:= 	FALSE;
ELSIF bVarExceptionAct THEN	
	bVarTKVardagAct:= 		FALSE;
	bVarTKVeckoslutAct:= 	FALSE;
	bVarHelgdagAktiv:= 		FALSE;
	bVarTKExceptionAct:=	TRUE;
END_IF

IF bVarTKVardagAct OR bVarTKVeckoslutAct OR bVarHelgdagAktiv OR bVarTKExceptionAct THEN
// Väljer korrekt offset i fallande prio om någon förskjutning ska ske
fbSel(
	diSelVal01:= 		diSPEveningReduction, 
	diSelVal02:= 		diSPWeekendReduction, 
	diSelVal03:= 		diSPHolidayReduction, 
	diSelVal04:= 		diSPExceptionReduction, 
	bEnabelVal01:= 		bVarTKVardagAct, 
	bEnabelVal02:= 		bVarTKVeckoslutAct, 
	bEnabelVal03:= 		bVarHelgdagAktiv, 
	bEnabelVal04:= 		bVarTKExceptionAct, 
	diOutPut=> 			diVarSelOutPut);
ELSE diVarSelOutPut:= 0;
	
END_IF

// Kör valt värde genom nedrampning
fbRamp(
	diInPutValue:= 		diVarSelOutPut, 
	diRampUpTime:= 		0, 
	diRampDownTime:= 	diDownRampTime, 
	diOutPutValue=> 	diVarOffsetValue, 
	bActive=> 			bRampTimeActive, 
	bUpDown=> 			);

// Larm för låg rumstemperatur	
IF diActualAverageRoomTemp <= diAllowedMinRoomTemp THEN
	bAlarmMinTemp:= TRUE; ELSE	
	bAlarmMinTemp:= FALSE;
END_IF

// PID som rampar ner förskjutning vid "kallt" i rum
fbPIDCascade(
	bEn:= 				bVarTKVardagAct OR bVarTKVeckoslutAct OR bVarHelgdagAktiv OR bVarTKExceptionAct,
	nPV:= 				diActualAverageRoomTemp,
	nSP:= 				diAllowedMinRoomTemp, 
	nP:= 				, 
	nI:= 				, 
	nD:= 				, 
	nDF:= 				, 
	nMAX:= 				diVarOffsetValue,
	nMIN:= 				0,
	nInitValue:= 		,
	nDeactValue:= 		diVarOffsetValue,
	bInvert:= 			,
	nY=> 				);


diKOHCalcOffset:= (diSystemCalcSetpoint - (diVarOffsetValue - fbPIDCascade.nY));




END_IF

END_IF
bAlarmBlocked:= 	bBlockKOHFunction;
bKOHBlocked:= 		bBlockKOHFunction;
diKOHCalcOffset:= 	diSystemCalcSetpoint;

END_FUNCTION_BLOCK

// ---- DUTs/Rampfunktion/FB_Ramp.TcPOU
FUNCTION_BLOCK FB_Ramp 
VAR_INPUT
	diInPutValue 		: DINT; // Inputvärde att rampa, skala 0.1
	diRampUpTime		: DINT; // Upprampning. Tidsenhet i sekunder, skala 0.1
	diRampDownTime		: DINT; // Upprampning. Tidsenhet i sekunder, skala 0.1
END_VAR         		
                		
VAR_OUTPUT      		
	diOutPutValue		: DINT; // Outputvärde som är rampat, samma skala som output
	bActive				: BOOL; // Rampning aktiv
	bUpDown				: BOOL; // TRUE = Värdet ökar, FALSE = Värde minskar
END_VAR         		
                		
VAR             		
	bVarInitiation		: BOOL; // Lokal variabel
	bVarRampAct			: BOOL; // Lokal variabel
	rVarInPut			: REAL; // Lokal variabel
	rVarRampUpTime		: REAL; // Lokal variabel
	rVarRampDownTime	: REAL; // Lokal variabel	
	rVarOutPut			: REAL; // Lokal variabel
	tVarSystemTime		: TIME; // Lokal variabel
	tVarLastTime		: TIME; // Lokal variabel
END_VAR

tVarSystemTime:= TIME();

IF diRampDownTime = 0 AND diRampUpTime = 0 THEN
	bVarRampAct   := FALSE;
	diOutPutValue := diInPutValue; ELSE
	bVarRampAct   := TRUE;
END_IF

rVarInPut 			:= TO_REAL (diInPutValue);
rVarRampUpTime 		:= TO_REAL (diRampDownTime);
rVarRampDownTime 	:= TO_REAL (diRampUpTime);

// Läser ur systemtiden i millisekunder
tVarSystemTime := tVarSystemTime - tVarLastTime;

IF NOT bVarInitiation THEN
	bVarInitiation 		:= TRUE;
	tVarLastTime 		:= tVarSystemTime;
	tVarSystemTime 		:= T#0S;
	rVarOutPut 			:= rVarInPut;
END_IF;

IF NOT bVarRampAct THEN
	rVarOutPut 			:= rVarInPut;
	bActive 			:= FALSE;

// Nedrampning	
ELSIF rVarOutPut > rVarInPut THEN
	rVarOutPut := rVarOutPut - TIME_TO_REAL(tVarSystemTime) * 0.001 * rVarRampUpTime;
	rVarOutPut := MAX(rVarInPut, rVarOutPut);

// Upprampning	
ELSIF rVarOutPut < rVarInPut THEN
	rVarOutPut := rVarOutPut + TIME_TO_REAL(tVarSystemTime) * 0.001 * rVarRampDownTime;
	rVarOutPut := MIN(rVarInPut, rVarOutPut);
END_IF;

diOutPutValue := TO_DINT (rVarOutPut);

// Sätter bActive och bUpDown
IF rVarOutPut < rVarInPut THEN
	bActive := TRUE;
	bUpDown := TRUE;
ELSIF rVarOutPut > rVarInPut THEN
	bActive := TRUE;
	bUpDown := FALSE;
ELSE
	bActive := FALSE;
END_IF;
tVarLastTime := tVarLastTime + tVarSystemTime;

END_FUNCTION_BLOCK

// ---- DUTs/Select/FB_Sel.TcPOU
FUNCTION_BLOCK FB_Sel
VAR_INPUT
	diSelVal01			: DINT;		// Ingång 0
	diSelVal02			: DINT;		// Ingång 1
	diSelVal03			: DINT;		// Ingång 2
	diSelVal04			: DINT;		// Ingång 3
	bEnabelVal01		: BOOL;		// Aktiverar diSelVal01
	bEnabelVal02		: BOOL;		// Aktiverar diSelVal02
	bEnabelVal03		: BOOL;		// Aktiverar diSelVal03
	bEnabelVal04		: BOOL;		// Aktiverar diSelVal04
END_VAR
VAR_OUTPUT
	diOutPut			: DINT;		// Aktiverat värde
END_VAR
VAR
END_VAR

IF bEnabelVal01 THEN
	diOutPut:=diSelVal01;
ELSIF bEnabelVal02 AND NOT bEnabelVal01 THEN
	diOutPut:=diSelVal02;
ELSIF bEnabelVal03 AND NOT bEnabelVal01 OR bEnabelVal02 THEN
	diOutPut:=diSelVal03;
ELSIF bEnabelVal04 AND NOT bEnabelVal01 OR bEnabelVal02 OR bEnabelVal03 THEN
	diOutPut:=diSelVal04;
ELSE
	diOutPut:=0;
END_IF

END_FUNCTION_BLOCK

// ---- DUTs/PID/FB_PID.TcPOU
FUNCTION_BLOCK FB_PID
VAR_INPUT
	bEn				: BOOL;				// Aktivera block
	nPV				: DINT; 			// Ärvärde
	nSP				: DINT; 			// Börvärde
	nP				: DWORD;			// P-faktor (OBS! Skala 1/100)
	nI				: DWORD;			// I-tid (s)
	nD				: DWORD;			// D-tid (s)
	nDF				: DWORD;			// Filter D-tid (s)
	nMAX			: DINT; 			// Maxbegränsning
	nMIN			: DINT; 			// Minbegränsning
	nInitValue		: DINT := 0;		// Initialt värde
	nDeactValue		: DINT := 0; 		// Värde vid inaktiverat block
	bInvert			: BOOL := FALSE; 	// Invertera funktion (T.ex. för Kyla)
END_VAR

VAR_OUTPUT
	nY				: DINT; 			// Styrsignal
END_VAR

VAR  
	DPart			: BOOL;
	FirstRun		: BOOL := TRUE;
	tx				: DWORD; 
	last			: DWORD;
	K 				: LREAL := 1.0;	
	KP 				: LREAL;
	TN 				: LREAL;
	TV 				: LREAL;
	TD 				: LREAL;
	Dd				: LREAL;
	Cd				: LREAL;
	YD				: LREAL;
	YD_1			: LREAL;
	E				: LREAL;
	E_1				: LREAL;
	Y				: LREAL;
	YI				: LREAL;
	LIM_L 			: LREAL;
	LIM_H 			: LREAL;
	E_last 			: LREAL;
	CycleTime		: LREAL;
	CycleTime_INT	: LREAL;
	Initvalue		: LREAL;	
	
	fbRTRIG			: R_TRIG;
END_VAR


CycleTime_INT	:= TO_LREAL(TwinCAT_SystemInfoVarList._TaskInfo[GETCURTASKINDEXEX()].CycleTime) / 10000;
CycleTime 		:= CycleTime_INT / 1000;
tx 				:= F_PLC_MS();

fbRTRIG(CLK := bEn);

IF NOT bEn OR FirstRun OR fbRTRIG.Q THEN
	
	KP 			:= 0.0;
	TN 			:= 0.0;
	TV 			:= 0.0;
	TD 			:= 0.0;
	Dd			:= 0.0;
	Cd			:= 0.0;
	E 	:= E_1	:= 0.0;
	YD	:= YD_1 := 0.0;
	DPart		:= FALSE;
	Initvalue	:= TO_LREAL(LIMIT((nMIN / 10), (nInitValue / 10), (nMAX / 10)));

ELSE
	// Save old values
	IF DPart THEN
		E_1	:= E;
		YD_1 := YD;
	END_IF
	
	KP		:= TO_LREAL(nP) / 1000;
	TN		:= TO_LREAL(nI) / 10;
	TV		:= TO_LREAL(nD) / 10;
	TD		:= TO_LREAL(nDF) / 10;
	LIM_L	:= TO_LREAL(nMin) / 10;
	LIM_H	:= TO_LREAL(nMax) / 10;

	IF Y < (LIM_L * 10) OR Y > (LIM_H * 10) THEN
		KP 			:= 0.0;
		TN 			:= 0.0;
		TV 			:= 0.0;
		TD 			:= 0.0;
		Dd			:= 0.0;
		Cd			:= 0.0;
		E 	:= E_1	:= 0.0;
		YD	:= YD_1 := 0.0;
		DPart		:= FALSE;
		Initvalue := LIMIT(LIM_L, (Y / 10), LIM_H); 
	END_IF
END_IF

// Invert function
IF NOT bInvert THEN
	E := (nSP - nPV);
ELSE
	E := (nPV - nSP);	
END_IF


// Integrator
IF tn = 0.0 OR NOT bEn THEN
	YI := 0.0;
ELSIF Y > (LIM_L * 10) AND Y < (LIM_H * 10) THEN
	YI := (E + E_LAST) * 0.5E-3 * DWORD_TO_LREAL(tx - last) * (K / TN) + YI;
	E_last := E;
END_IF
last := tx;


// Add up integrator and linear part 
Y := KP * (E + YI);


// D-part
IF TV > 0.0 AND TD > 0.0 THEN
	Dd := ((KP * TV) / (TD + CycleTime / 2.0));
	Cd := ((TD - CycleTime / 2.0) / (TD + CycleTime / 2.0));
	DPart := TRUE;
ELSE
	Dd := 0.0;
	Cd := 0.0;
	DPart := FALSE;
END_IF
	
// YD-part 
IF DPart THEN
	YD	:=  (Cd * YD_1 + Dd * (E - E_1));
ELSE
	YD	:= 0.0;
END_IF
																																		

// Add differential part, initvalue and limit output Y 
Y := LIMIT((LIM_L * 10), ((Y + YD + Initvalue) * 10), (LIM_H * 10));


// Output
IF NOT bEn THEN
	nY := nDeactValue;
ELSE
	nY := TO_DINT(Y);
END_IF

FirstRun := FALSE;

END_FUNCTION_BLOCK

// ---- DUTs/Helgdag/Old/POU_EasterDay.TcPOU
PROGRAM POU_EasterDay
VAR
	fbSystemTime 				: FB_SystemTime;
	
    iYear 						: INT; (* Ange året här *)
    iMonth						: INT;
	iDay						: INT;
    iEastermDayOfYear			: INT;     (* Påskdagens dagnummer i året *)
    isLeapYear 					: BOOL;   (* Flagga för skottår *)	
	stSystemTime				: TIMESTRUCT;
    arrMonthDays 				: ARRAY[1..12] OF INT := [31,28,31,30,31,30,31,31,30,31,30,31]; (* Dagar per månad *)
    iDayOfYear					: INT;
	dActDate					: DATE_AND_TIME; 
    (* Variabler för Gauss algoritm *)
    a, b, c, d, e, f, g, h, i, k, L, m, n : INT;
	iDayOfWeek					: INT;
	
	iVarHalloweenDay			: INT;
	iVarMidsommardagen 			: INT;
	iVarMidsommardagen1			: INT;
	iVarMidsommardagenDayOfWeek	: INT;
	iVarDayOfYearCristmas		: INT;
	iVarDayForstamaj			: INT;
	iVarNationaldag				: INT;
	iVarJuldagen				: INT;
	
	iLangfredag					: INT;
 	iSkartorsdag				: INT;
	iPaskDagen					: INT;
 	iPaskafton					: INT;
 	iAnnanDagPask				: INT;
	iKristihimmel				: INT;
	iPingstAfton				: INT;
	iPingstDagen				: INT;
	iMidsommarDagen				: INT;
	iMidsommarAfton				: INT;
	iHalloween					: INT;
	iJulafton					: INT;
	iJuldagen					: INT;
	iAnnandagjul				: INT;
	iTrettondag					: INT;
    iNyarsafton					: INT;	
    iNyarsdagen					: INT;	
    iForstamaj					: INT;		
    iNationaldag				: INT;
	
	bLangfredag					: BOOL;
	bSkartorsdag				: BOOL;
	bPaskDagen					: BOOL;
    bPaskafton					: BOOL;
    bAnnanDagPask				: BOOL;
    bKristihimmel				: BOOL;
    bPingstAfton				: BOOL;
    bPingstDagen				: BOOL;
    bMidsommarDagen				: BOOL;
    bMidsommarAfton				: BOOL;
    bHalloween					: BOOL;
    bJulafton					: BOOL;
    bJuldagen					: BOOL;
    bAnnandagjul				: BOOL;
    bTrettondag					: BOOL;
    bNyarsafton					: BOOL;
    bNyarsdagen					: BOOL;
    bForstamaj					: BOOL;
    bNationaldag				: BOOL;

	
END_VAR

fbSystemTime();
iDayOfYear:=fc_Day_Of_Year(IDATE:=TO_DATE (fbSystemTime.dtSystemTime));
iYear:= DWORD_TO_INT(fbSystemTime.nYear);
iDayOfWeek:= DWORD_TO_INT(fbSystemTime.nDay);


// Gauss algoritm för att räkna ut påskdagen
a := iYear MOD 19;
b := iYear / 100;
c := iYear MOD 100;
d := b / 4;
e := b MOD 4;
f := (b + 8) / 25;
g := (b - f + 1) / 3;
h := (19 * a + b - d - g + 15) MOD 30;
i := c / 4;
k := c MOD 4;
L := (32 + 2 * e + 2 * i - h - k) MOD 7;
m := (a + 11 * h + 22 * L) / 451;
n := (h + L - 7 * m + 114);
iMonth := n / 31;
iEastermDayOfYear := (n MOD 31) + 1;

// Kontrollera om året är skottår
IF (iYear MOD 4 = 0 AND iYear MOD 100 <> 0) OR (iYear MOD 400 = 0) THEN
    isLeapYear := TRUE;
    arrMonthDays[2] := 29; // Februari har 29 dagar i skottår
ELSE
    isLeapYear := FALSE;
END_IF

// Beräkna årets dag för påskdagen
iEastermDayOfYear := iDay; // Startvärde
FOR i := 1 TO iMonth - 1 DO
    iEastermDayOfYear := iEastermDayOfYear + arrMonthDays[i]; // Addera dagar i tidigare månader
END_FOR

// Beräkna årets dag för 31 oktober, Halloween
iVarHalloweenDay := 31; // Startvärde för Halloweens dag i oktober
FOR i := 1 TO 9 DO // Loopar igenom månaderna januari-september
    iVarHalloweenDay := iVarHalloweenDay + arrMonthDays[i]; // Addera dagar i tidigare månader
END_FOR

IF isLeapYear THEN
    iVarHalloweenDay := iVarHalloweenDay + 1;
END_IF

// Beräkna veckodag för 20 juni, midsommardagen
// Formel för veckodag (Zeller's Congruence)
iVarMidsommardagenDayOfWeek := (20 + ((13 * 6 + 1) / 5) + (iYear MOD 100) + ((iYear MOD 100) / 4) + ((iYear / 100) / 4) - (2 * (iYear / 100))) MOD 7;
IF iVarMidsommardagenDayOfWeek < 0 THEN
    iVarMidsommardagenDayOfWeek := iVarMidsommardagenDayOfWeek + 7; // Hantera negativa veckodagar
END_IF

// Hitta första lördagen efter 20 juni
iVarMidsommardagen := 20 + ((6 - iVarMidsommardagenDayOfWeek) MOD 7) + 1;

// Beräkna årets dag för midsommardagen
iVarMidsommardagen1 := iVarMidsommardagen;
FOR i := 1 TO 5 DO // Loopar igenom månaderna januari-maj
    iVarMidsommardagen1 := iVarMidsommardagen1 + arrMonthDays[i]; //Addera dagar i tidigare månader
END_FOR

// Beräknar årets dag för 25 december
iVarDayOfYearCristmas := 24; // Startvärde för juldagen
FOR i := 1 TO 11 DO // Loopar igenom månaderna januari-november
    iVarDayOfYearCristmas := iVarDayOfYearCristmas + arrMonthDays[i]; // Addera dagar i tidigare månader
END_FOR

IF isLeapYear THEN
    iVarDayOfYearCristmas := iVarDayOfYearCristmas + 1;
END_IF

// Beräknar årets dag för 1 maj
iVarDayForstamaj := 0; // Startvärde för 1 maj
FOR i := 1 TO 4 DO // Loopar igenom månaderna januari-april *)
    iVarDayForstamaj := iVarDayForstamaj + arrMonthDays[i]; //Addera dagar i tidigare månader
END_FOR

IF isLeapYear THEN
    iVarDayForstamaj := iVarDayForstamaj + 1;
END_IF

// Beräkna sveriges nationaldag
iVarNationaldag := 5; // Startvärde för 6 juni
FOR i := 1 TO 5 DO // Loopar igenom månaderna januari-maj
    iVarNationaldag := iVarNationaldag + arrMonthDays[i]; // Addera dagar i tidigare månader
END_FOR
IF isLeapYear THEN
    iVarNationaldag := iVarNationaldag + 1;
END_IF

// Ger var värde för resp. dag
iLangfredag 		:= iEastermDayOfYear - 2;
iSkartorsdag	 	:= iEastermDayOfYear - 3;
iPaskDagen			:= iEastermDayOfYear;
iPaskafton 			:= iEastermDayOfYear - 1; 
iAnnanDagPask 		:= iEastermDayOfYear + 1; 
iKristihimmel 		:= iEastermDayOfYear + 39; 
iPingstAfton		:= iEastermDayOfYear + 48; 
iPingstDagen		:= iEastermDayOfYear + 49;
iMidsommarDagen		:= iVarMidsommardagen1;
iMidsommarAfton		:= iVarMidsommardagen1 - 1;
iHalloween			:= iVarHalloweenDay;
iJulafton			:= iVarDayOfYearCristmas - 1;
iJuldagen			:= iVarDayOfYearCristmas;
iAnnandagjul		:= iVarDayOfYearCristmas + 1;
iTrettondag			:= 6;
iNyarsafton			:= iVarDayOfYearCristmas + 6;
iNyarsdagen			:= 1; 
iForstamaj			:= iVarDayForstamaj;
iNationaldag		:= iVarNationaldag;

// Sätter bool för resp. dag
bLangfredag 		:= (iDayOfYear = (iLangfredag));
bSkartorsdag	 	:= (iDayOfYear = (iSkartorsdag));
bPaskDagen			:= (iDayOfYear = (iPaskDagen));
bPaskafton 			:= (iDayOfYear = (iPaskafton));
bAnnanDagPask 		:= (iDayOfYear = (iAnnanDagPask));
bKristihimmel 		:= (iDayOfYear = (iKristihimmel));
bPingstAfton		:= (iDayOfYear = (iPingstAfton));
bPingstDagen		:= (iDayOfYear = (iPingstDagen));
bMidsommarDagen		:= (iDayOfYear = (iMidsommarDagen));
bMidsommarAfton		:= (iDayOfYear = (iMidsommarAfton));
bHalloween			:= (iDayOfYear = (iHalloween));
bJulafton			:= (iDayOfYear = (iJulafton));
bJuldagen			:= (iDayOfYear = (iJuldagen));
bAnnandagjul		:= (iDayOfYear = (iAnnandagjul));
bTrettondag			:= (iDayOfYear = (iTrettondag));
bNyarsafton			:= (iDayOfYear = (iNyarsafton));
bNyarsdagen			:= (iDayOfYear = (iNyarsdagen));
bForstamaj			:= (iDayOfYear = (iForstamaj));
bNationaldag		:= (iDayOfYear = (iNationaldag));

END_PROGRAM

// ---- DUTs/Helgdag/Old/FB_SwedishHolidaysOLD.TcPOU
FUNCTION_BLOCK FB_SwedishHolidaysOLD
VAR_INPUT
    iYear 					: INT; // Aktuellt år
    dtCurrentDate 			: DATE_AND_TIME; // Dagens datum
END_VAR

VAR_OUTPUT
   	bMaundyThursday			: BOOL; // Skärtorsdag
   	bGoodFriday 			: BOOL; // Långfredag
   	bEasterSaturday			: BOOL; // Påskafton
   	bEasterSunday 			: BOOL; // Påskdagen
   	bEasterMonday 			: BOOL; // Annandag påsk
	bAscensionDay			: BOOL; // Kristihimmelsfärds dag
	
	bJulAfton				: BOOL; // Julafton
	bJulDagen				: BOOL; // Juldagen
	bAnnandagJul			: BOOL; // Annandag jul
	bTrettonDagJul			: BOOL; // Trettondagsjul
	
	bNyArsAfton				: BOOL; // Nyårsafton
	bNyArsDagen				: BOOL; // Nyårsdagen
	
	bPingstAfton			: BOOL; // Pingstafton
	bPingstDagen			: BOOL; // Pingstdagen
	
	bMidsommarafton			: BOOL; // Midsommarafton
	bMidsommarDagen 		: BOOL; // Midsommardagen
	bHalloween 				: BOOL; // Alla helgons dag, Halloween
	
	bForstaMaj				: BOOL; // Första Maj
	bSverigesNationaldag 	: BOOL; // Sveriges nationaldag
	
	bAnyHolidayActive		: BOOL; // Någon helgdag är aktiv
	
END_VAR

VAR
    iA, iB, iC, iD, iE, iMonth, iDay : INT;
    udiGoodFriday			: UDINT;
	udiMaundyThursday		: UDINT;
	udiEasterSaturday		: UDINT;
	udiEasterMonday			: UDINT;
	udiAscensionDay			: UDINT;
	udiPingstAfton			: UDINT;
	udiPingstDagen			: UDINT;
	udiMidsommardagen		: UDINT;
	stPaskdagen 			: TIMESTRUCT;
	stSystemTime			: TIMESTRUCT;
	stMidsommarAfton		: TIMESTRUCT;
	stMidsommarDagen		: TIMESTRUCT;
	stHalloween				: TIMESTRUCT;

	iForMidsommarday		: INT; // forloop midsommardagen 20-25 (23:59)
	dtVarMidsommar 			: DATE_AND_TIME; // lokal var
	stVarMidsommarCalc 		: TIMESTRUCT; // Lokal va
	
	iForHalloween			: INT; // forloop halloween 31-06 månadsbrytr
	stVarHalloweenCalc		: TIMESTRUCT;
	bVarHalloween			: BOOL; // Lokal var
	dtVarHalloween			: DATE_AND_TIME; 
	
	iVarSummaHelgdag		: INT; // forloop summa helgdag
	arrHelgDag				: ARRAY [1..19] OF BOOL;
	
	stAscensionDay			: TIMESTRUCT;
	stPingstDagen			: TIMESTRUCT;
END_VAR

// Beräkning av påskdagen med Gauss' algoritm
iA := iYear MOD 19;
iB := iYear MOD 4;
iC := iYear MOD 7;
iD := (19 * iA + 24) MOD 30;
iE := ((2 * iB) + (4 * iC) + (6 * iD) + 5) MOD 7;
iDay := 22 + iD + iE; // Påskdagen i mars eller april
stSystemTime:= DT_TO_SYSTEMTIME(dtCurrentDate);

IF iDay > 31 THEN
    iMonth := 4; ELSE 
    iMonth := 3; 
END_IF;

IF iDay <= 31 THEN
	stPaskdagen.wMonth := 3;
	stPaskdagen.wDay := INT_TO_WORD(iDay); ELSE
	stPaskdagen.wMonth := 4;
	stPaskdagen.wDay := INT_TO_WORD(iDay - 31);
END_IF

IF stPaskdagen.wMonth = 4 AND stPaskdagen.wDay = 26 THEN
	stPaskdagen.wDay := 19;
END_IF

IF stPaskdagen.wMonth = 4 AND stPaskdagen.wDay = 25 AND iD = 28 AND iE = 6 AND iA > 10 THEN
	stPaskdagen.wDay := 18;
END_IF

// Beräknar midsommar
stMidsommarAfton.wYear := stSystemTime.wYear;
stMidsommarAfton.wMonth := 6;
FOR iForMidsommarday := 20 TO 26 DO
	stMidsommarAfton.wDay := INT_TO_WORD(iForMidsommarday);
	dtVarMidsommar := SYSTEMTIME_TO_DT(stVarMidsommarCalc);
	stVarMidsommarCalc := DT_TO_SYSTEMTIME(dtVarMidsommar);

IF stVarMidsommarCalc.wDayOfWeek = 5 THEN
	stMidsommarAfton := stVarMidsommarCalc;
END_IF

END_FOR

// Beräknar halloween
stVarHalloweenCalc.wYear := stSystemtime.wYear;
stVarHalloweenCalc.wMonth := 11;
bVarHalloween := FALSE;
FOR iForHalloween := 1 TO 6 DO
	stVarHalloweenCalc.wDay := INT_TO_WORD(iForHalloween);
	dtVarHalloween := SYSTEMTIME_TO_DT(stVarHalloweenCalc);
	stVarHalloweenCalc := DT_TO_SYSTEMTIME(dtVarHalloween);
	
	IF stVarHalloweenCalc.wDayOfWeek = 6 THEN
		stHalloween := stVarHalloweenCalc;
		bVarHalloween := TRUE;
		EXIT;
		ELSIF stVarHalloweenCalc.wDay = 6 AND NOT bVarHalloween THEN
			stHalloween.wMonth := 10;
			stHalloween.wDay := 31;			
	END_IF
END_FOR

// Beräknar kristi himmelsfärd
IF stPaskdagen.wDay > 22 THEN
	stAscensionDay.wMonth := stPaskdagen.wMonth + 2;
	stAscensionDay.wDay := stPaskdagen.wDay - 22;
	ELSIF stPaskdagen.wMonth = 3 THEN
		stAscensionDay.wDay := stPaskdagen.wDay + 8;
	ELSE stAscensionDay.wDay := stPaskdagen.wDay + 9;
END_IF


// Beräknar pingstdagen
IF stAscensionDay.wMonth = 4 THEN
	stPingstDagen.wMonth := 5;
	stPingstDagen.wDay := 10;
END_IF

IF stAscensionDay.wMonth = 5 AND stAscensionDay.wMonth > 20 THEN
	stPingstDagen.wMonth := 6;
	stPingstDagen.wDay := stAscensionDay.wDay - 20;
	ELSIF stAscensionDay.wMonth = 5 AND stAscensionDay.wMonth <= 20 THEN
			stPingstDagen.wMonth := 5;
			stPingstDagen.wDay := stAscensionDay.wDay + 10;
				ELSE stPingstDagen.wMonth := 6;
				stPingstDagen.wDay := stAscensionDay.wDay + 10;
END_IF

// Beräkna de andra helgdagarna
udiGoodFriday 		:= stPaskdagen.wDay - 2;
udiMaundyThursday 	:= stPaskdagen.wDay - 3;
udiEasterSaturday 	:= stPaskdagen.wDay - 1;
udiEasterMonday 	:= stPaskdagen.wDay + 1;
udiAscensionDay 	:= stPaskdagen.wDay + 39;
udiPingstAfton		:= stPaskdagen.wDay + 48;
udiPingstDagen		:= stPaskdagen.wDay + 49;
udiMidsommarDagen	:= stMidsommarAfton.wDay + 1;

// Sätter utgångar

// Skärtorsdag
IF stSystemTime.wMonth = stPaskdagen.wMonth AND stSystemTime.wDay = udiMaundyThursday THEN
	bMaundyThursday := TRUE; ELSE
	bMaundyThursday := FALSE;
END_IF

// Långfredag
IF stSystemTime.wMonth = stPaskdagen.wMonth AND stSystemTime.wDay = udiGoodFriday THEN
	bGoodFriday := TRUE; ELSE
	bGoodFriday := FALSE;
END_IF

// Påskafton
IF stSystemTime.wMonth = stPaskdagen.wMonth AND stSystemTime.wDay = udiEasterSaturday THEN
	bEasterSaturday := TRUE; ELSE
	bEasterSaturday := FALSE;
END_IF

// Påskdagen
IF stSystemTime.wMonth = stPaskdagen.wMonth AND stSystemTime.wDay = stPaskdagen.wDay THEN
	bEasterSunday := TRUE; ELSE
	bEasterSunday := FALSE;
END_IF

// Annandag påsk
IF stSystemTime.wMonth = stPaskdagen.wMonth AND stSystemTime.wDay = udiEasterMonday THEN
	bEasterMonday := TRUE; ELSE
	bEasterMonday := FALSE;
END_IF

// Kristi himmelsfärd
IF stSystemTime.wMonth = stPaskdagen.wMonth +1  AND stSystemTime.wDay  = stPaskdagen.wDay +9 THEN
	bAscensionDay := TRUE; ELSE
	bAscensionDay := FALSE;
END_IF

// Julafton
IF stSystemTime.wMonth = 12 AND stSystemTime.wDay = 24 THEN
	bJulAfton:= TRUE; ELSE
	bJulAfton:= FALSE;
END_IF

// Juldagen
IF stSystemTime.wMonth = 12 AND stSystemTime.wDay = 25 THEN
	bJulDagen:= TRUE; ELSE
	bJulDagen:= FALSE;
END_IF

// Annandag jul
IF stSystemTime.wMonth = 12 AND stSystemTime.wDay = 26 THEN
	bAnnandagJul:= TRUE; ELSE
	bAnnandagJul:= FALSE;
END_IF

// Trettondag jul
IF stSystemTime.wMonth = 1 AND stSystemTime.wDay = 6 THEN
	bTrettonDagJul:= TRUE; ELSE
	bTrettonDagJul:= FALSE;
END_IF

// Nyårsafton
IF stSystemTime.wMonth = 12 AND stSystemTime.wDay = 31 THEN
	bNyArsAfton:= TRUE; ELSE
	bNyArsAfton:= FALSE;
END_IF

// Nyårsdagen
IF stSystemTime.wMonth = 1 AND stSystemTime.wDay = 1 THEN
	bNyArsDagen:= TRUE; ELSE
	bNyArsDagen:= FALSE;
END_IF

// Pingstafton
IF stSystemTime.wMonth = stPingstDagen.wMonth AND stSystemTime.wDay = stPingstDagen.wDay -1 THEN
	bPingstAfton := TRUE; ELSE
	bPingstAfton := FALSE;
END_IF

// Pingstdagen
IF stSystemTime.wMonth = stPaskdagen.wMonth +1 AND stSystemTime.wDay = stPingstDagen.wDay THEN
	bPingstAfton := TRUE; ELSE
	bPingstAfton := FALSE;
END_IF

// Midsommarafton
IF stSystemTime.wMonth = stMidsommarAfton.wMonth AND stSystemTime.wDay = stMidsommarAfton.wDay THEN
	bMidsommarafton:= TRUE; ELSE
	bMidsommarafton:= FALSE;
END_IF

// Midsommardagen
IF stSystemTime.wMonth = stMidsommarDagen.wMonth AND stSystemTime.wDay = stMidsommarDagen.wDay THEN
	bMidsommarDagen:= TRUE; ELSE
	bMidsommarDagen:= FALSE;
END_IF

// Halloween
IF stSystemTime.wMonth = stHalloween.wMonth AND stSystemTime.wDay = stHalloween.wDay THEN
	bHalloween:= TRUE; ELSE
	bHalloween:= FALSE;
END_IF

// Första maj
IF stSystemTime.wMonth = 5 AND stSystemTime.wDay = 1 THEN
	bForstaMaj:= TRUE; ELSE
	bForstaMaj:= FALSE;
END_IF

// Sveriges nationaldag
IF stSystemTime.wMonth = 6 AND stSystemTime.wDay = 6 THEN
	bSverigesNationaldag:= TRUE; ELSE
	bSverigesNationaldag:= FALSE;
END_IF


arrHelgDag[1]:= bMaundyThursday;
arrHelgDag[2]:= bGoodFriday;
arrHelgDag[3]:= bEasterSaturday;
arrHelgDag[4]:= bEasterSunday;
arrHelgDag[5]:= bEasterMonday;
arrHelgDag[6]:= bAscensionDay;
arrHelgDag[7]:= bJulAfton;
arrHelgDag[8]:= bJulDagen;
arrHelgDag[9]:= bAnnandagJul;
arrHelgDag[10]:= bTrettonDagJul;
arrHelgDag[11]:= bNyArsAfton;
arrHelgDag[12]:= bNyArsDagen;
arrHelgDag[13]:= bPingstAfton;
arrHelgDag[14]:= bPingstDagen;
arrHelgDag[15]:= bMidsommarafton;
arrHelgDag[16]:= bMidsommarDagen;
arrHelgDag[17]:= bHalloween;
arrHelgDag[18]:= bForstaMaj;
arrHelgDag[19]:= bSverigesNationaldag;

iVarSummaHelgdag := 1;
FOR iVarSummaHelgdag := 1 TO 19 DO
	IF arrHelgDag[iVarSummaHelgdag] THEN
	bAnyHolidayActive:= TRUE;
	EXIT;
	ELSE bAnyHolidayActive:= FALSE;
		
	END_IF
END_FOR

END_FUNCTION_BLOCK

// ---- DUTs/Scale/FB_Scale.TcPOU
FUNCTION_BLOCK FB_Scale
VAR_INPUT	
	diInPutToScale			:DINT; // Värde som ska skalas
	diX0StarterValScaled	:DINT; // Startvärde, tex 0
	diX1EndValScaled		:DINT; // Slutvärde, tex 1000
	diY0StartOut			:DINT; // Startvärde skalat
	iY1EndOut				:DINT; // Slutvärde skalat
END_VAR
VAR_OUTPUT
	diOutPutVal				:DINT; // Utvärde
END_VAR

IF diX1EndValScaled > 0 AND diX1EndValScaled > diX0StarterValScaled  THEN 
	diOutPutVal := (diInPutToScale - diX0StarterValScaled) * (iY1EndOut - diY0StartOut) / (diX1EndValScaled - diX0StarterValScaled) + iY1EndOut;
	ELSE diOutPutVal := 0;
END_IF

END_FUNCTION_BLOCK
